FUNCTION_BLOCK T_MaintenanceMode IMPLEMENTS I_PackMLMode
VAR
	
END_VAR

END_FUNCTION_BLOCK

(* stored: Version 1.1.0.1, ProductVersion 3.1.4024.12
   POU T_MaintenanceMode: Id {1b9b4d90-2c46-4764-9e9a-b59cfa023b3b}, SpecialFunc None *)
